TYPE E_S19RecordState :
(
	Undefined := 0,
	Valid,
	BlockEnd,
	NotComplete,
	CRC_Error,
	Line_Error
)USINT;
END_TYPE

(* stored: Version 1.1.0.1, ProductVersion 3.1.0.25
   DUT E_S19RecordState: Id {029c4b7f-dbe1-4688-9329-e65868e20ab6} *)
